# B&R Automation Studio project rand
Automation Studio 

## Logical view

### Program Logical/rand1 (ANSIC)

#### rand1Cyclic.c - Cyclic code
```c
/********************************************************************
 * COPYRIGHT -- Bernecker + Rainer
 ********************************************************************
 * Program: rand1
 * File: rand1Cyclic.c
 * Author: vancurar
 * Created: May 22, 2014
 ********************************************************************
 * Implementation of program rand1
 ********************************************************************/

#include <bur/plctypes.h>
#include <stdlib.h>

#ifdef _DEFAULT_INCLUDES
	#include <AsDefault.h>
#endif

void _INIT rand1Init(void)
{
	/* generátor náhodných čísel je třeba zinicializovat aby se generovala vždy různá posloupnost čísel */
	DTGetTime_0.enable = 1;
	DTGetTime(&DTGetTime_0);

	srand(DTGetTime_0.DT1);

	/* následující řádek je pouze pro kontrolu, zda je první je první náhodé číslo vždy jiné */
	firstNumber = rand();
}

void _CYCLIC rand1Cyclic(void)
{
	/* zavoláním tohoto řádku se do "r" přiřad9 náhodné číslo v rozsahu 1 až 5 */
	r = 1 + rand() % 5;
}
```

#### rand1.var - Local variables
```iecst
(********************************************************************
 * COPYRIGHT -- Bernecker + Rainer
 ********************************************************************
 * Program: rand1
 * File: rand1.var
 * Author: vancurar
 * Created: May 22, 2014
 ********************************************************************
 * Local variables of program rand1
 ********************************************************************)
VAR
	DTGetTime_0 : DTGetTime := (0);
	firstNumber : INT := 0;
	r : INT := 0;
END_VAR
```
